// ---- POUs/MSG/Visualization.TcVIS
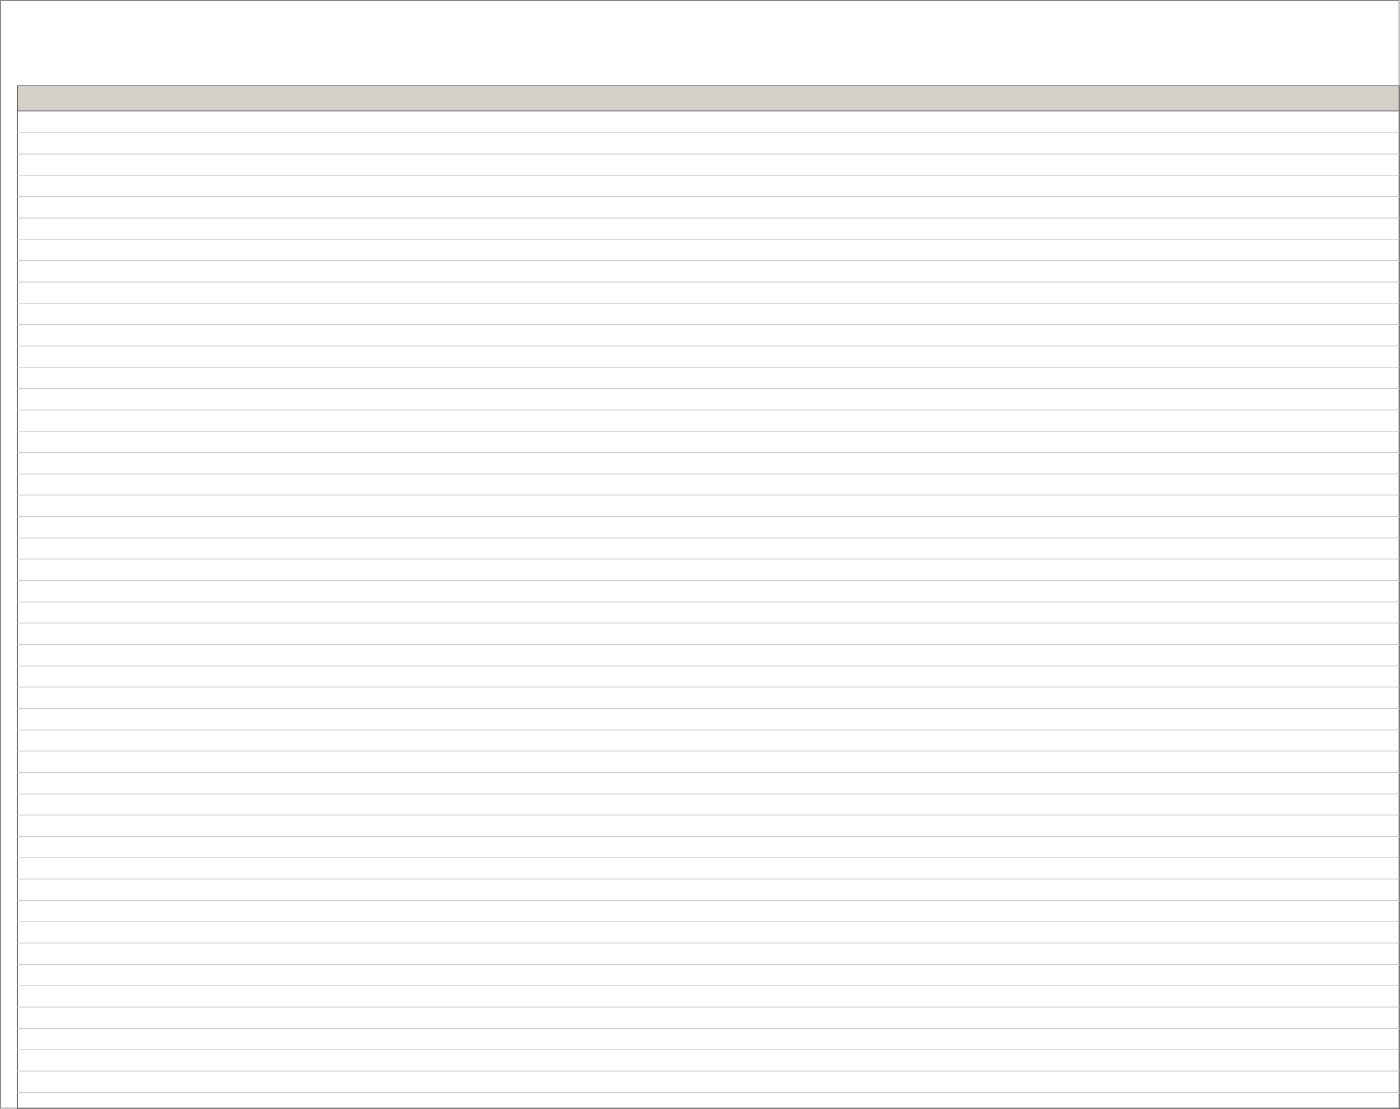
VISUALIZATION Visualization  // 1640x1300
    Table (20,100 1620x1200), data array: p_Data.VisuList
        p1128707560: GVL_AXIS_CTRL.gciMaxMessage
        p3854506369: p_Data.VisuList[INDEX].eType
        p1892666644: p_Data.VisuList[INDEX].eDevice
        p338671338: p_Data.VisuList[INDEX].eSubdevice
        p2170511999: p_Data.VisuList[INDEX].iErrorNumber
        p3723444502: p_Data.VisuList[INDEX].tTime
        p1218418051: p_Data.VisuList[INDEX].sText
END_VISUALIZATION
